FUNCTION_BLOCK FB_ValueDeviation IMPLEMENTS I_ValueDeviation, I_ValueDeviationLimited

VAR
	_delayDeviation		: Tc2_Standard.TON;
	_value				: ST_Value;
	_status				: E_ValueDeviationStatus;
	_maxDeviation		: T_ControllerValue;
	_enable				: BOOL;
	_activationDelay	: TIME;
END_VAR

IF _enable THEN
	_delayDeviation(
	IN := ABS(_value.Setpoint - _value.Actual) > ABS(_maxDeviation), 
	PT := _activationDelay);
ELSE
	_delayDeviation(IN := FALSE);
END_IF

IF _delayDeviation.Q THEN
	_status := E_ValueDeviationStatus.NOK;
ELSE
	_status := E_ValueDeviationStatus.OK;
END_IF

{attribute 'monitoring':='call'}
(* Gets or sets the activation delay, before the deviation error is activated*)
PROPERTY ActivationDelay : TIME
GET
ActivationDelay := _activationDelay;
END_GET
SET
_activationDelay := ActivationDelay;
END_SET
END_PROPERTY

{attribute 'monitoring':='call'}
PROPERTY Enable : BOOL
GET
Enable := _enable;
END_GET
SET
_enable := Enable;
END_SET
END_PROPERTY

{attribute 'monitoring':='call'}
PROPERTY MaxDeviation : REAL
GET
MaxDeviation := _maxDeviation;
END_GET
SET
_maxDeviation := MaxDeviation;
END_SET
END_PROPERTY

{attribute 'monitoring':='call'}
PROPERTY Status : E_ValueDeviationStatus
GET
Status := _status;
END_GET
END_PROPERTY

{attribute 'monitoring':='call'}
PROPERTY Value : REFERENCE TO ST_Value
GET
Value REF= _value;
END_GET
END_PROPERTY

END_FUNCTION_BLOCK

(* stored: Version 1.1.0.1, ProductVersion 3.1.4024.14
   POU FB_ValueDeviation: Id {c5ff19cb-11c2-0f72-212a-d933426c76a3}, SpecialFunc None
   Property ActivationDelay: Id {f6da7b17-0167-0ecf-0d12-e0217755d6d2}
   Get Get: Id {e55c933f-15e8-0e15-15ab-9ff66dd74ba8}
   Set Set: Id {f7695020-3f03-0a2b-3624-34c9d0689f53}
   Property Enable: Id {c18448c6-0347-06e4-2819-263c70e9f861}
   Get Get: Id {cfd4c918-6d3c-0522-1331-fce8faf72d4d}
   Set Set: Id {8e0a88df-9fd2-018c-339c-bcd28bd8736e}
   Property MaxDeviation: Id {d1002e23-4697-0a96-0366-6fecf8049e2c}
   Get Get: Id {9c431166-f7de-07f8-1d09-3b35f84faaf4}
   Set Set: Id {bbe83b6a-05c5-0c9b-2a14-95fe7c29f4ff}
   Property Status: Id {1bc020c4-ab28-03f6-22c6-5e31f8c03b04}
   Get Get: Id {c0e28e53-20fd-0bb9-0c93-60722768b814}
   Property Value: Id {d7c3bcec-ec7e-089a-26c7-6a9b1f2a8aad}
   Get Get: Id {75356649-6e51-0d93-0d31-54fba61d16b6} *)
